FUNCTION_BLOCK FourStateDeviceControl EXTENDS FourStateDevice
VAR
	OnOffCmd AT%I* : BOOL;
	
	App_OnOff: BOOL;
	App_FanSpeed: INT;
	
	rtOnOffCmd: R_TRIG;
	rtApp_OnOff: R_TRIG;
	FanSpeed_prev: INT;
END_VAR


	rtOnOffCmd(CLK:= OnOffCmd, Q=> );
	rtApp_OnOff(CLK:= App_OnOff, Q=> );

	IF rtOnOffCmd.Q OR rtApp_OnOff.Q THEN
		IF Status <> 0 THEN
			Off();
		ELSE		
			On();	
		END_IF
	END_IF

	CASE App_FanSpeed OF
		
		0: 	FanSpeed_prev	:=	App_FanSpeed;
		
		1: 	
			IF (FanSpeed_prev <> App_FanSpeed) THEN
				FanSpeed_prev	:=	App_FanSpeed;
				State_1();
			END_IF			
			
		2: 	
			IF (FanSpeed_prev <> App_FanSpeed) THEN
				FanSpeed_prev	:=	App_FanSpeed;
				State_2();
			END_IF			
			
		3: 	
			IF (FanSpeed_prev <> App_FanSpeed) THEN
				FanSpeed_prev	:=	App_FanSpeed;
				State_3();
			END_IF			
			
		4: 	
			IF (FanSpeed_prev <> App_FanSpeed) THEN
				FanSpeed_prev	:=	App_FanSpeed;
				State_4();
			END_IF			
			
	END_CASE

END_FUNCTION_BLOCK

(* stored: Version 1.1.0.1, ProductVersion 3.1.4024.13
   POU FourStateDeviceControl: Id {260d3c92-a109-450c-a1a7-539ddcb9daba}, SpecialFunc None *)
